FUNCTION_BLOCK TestAxis2 EXTENDS FB_ComponentBase
VAR
	AxisSPT : FB_BasicAxis;
	State 	: INT;
END_VAR

METHOD PUBLIC CyclicLogic
VAR	

END_VAR
SUPER^.CyclicLogic();
END_METHOD

METHOD PROTECTED Initialize : BOOL;
SUPER^.Initialize();
END_METHOD

METHOD MoveAxis
      AxisSPT.CyclicLogic();

IF SafetyGlobalVariableList.SAFETY_Permission = TRUE THEN

	CASE State OF
		
	00:
		IF AxisSPT.Enable() THEN
			State := State + 10;
		END_IF
	10:
		IF AxisSPT.Enabled THEN
			AxisSPT.MoveVelocity( -5, TRUE);	
		
			IF IO.DI4 = TRUE THEN
				AxisSPT.Home();
				State := State + 10;
			END_IF
		END_IF

	
	20:
		AxisSPT.Velocity := 10;
		IF AxisSPT.MoveAbsolute(5000, FALSE) THEN
			State := State + 10;
		END_IF

	30:
		IF NOT AxisSPT.Busy THEN
			State := State + 10;
		END_IF

	40:
		AxisSPT.Trace('****Done****'); 

	50:
		//

	END_CASE

END_IF
END_METHOD

END_FUNCTION_BLOCK

(* stored: Version 1.1.0.1, ProductVersion 3.1.4024.15
   POU TestAxis2: Id {c4d1aeed-ad07-48ee-832a-cb3f45f1be38}, SpecialFunc None
   Method CyclicLogic: Id {add4678a-922e-4e32-840c-f1dbbb6cbc7b}
   Method Initialize: Id {373c7236-707d-4500-91b5-e3c3f285aa21}
   Method MoveAxis: Id {60e94f90-6698-4c2d-a40d-761d438c97f6} *)
